# EPICS autosave request: VatLeakValve590/VATLeakValve590series_settings.req
$(device):SETF2IGAIN
$(device):SETF2PGAIN
$(device):SETPOSITIONLIMIT
$(device):SETPRESSURELIMIT
$(device):SETVALVESPEED
